FUNCTION IS_CTRL : BOOL
VAR_INPUT
	STR : STRING(STRING_LENGTH);
END_VAR
VAR
	L: INT;
	pt : POINTER TO BYTE;
	pos: INT;
END_VAR

(*
version 1.1	29. mar 2008
programmer 		kurt
tested by		hugo

IS_CTRL testet ob in einem string nur Steuerzeichen (Char < 32) vorkommen.

*)

PT := ADR(str);
L := LEN(str);
FOR pos := 1 TO L DO
	IF NOT (ISC_CTRL(pt^)) THEN
		IS_CTRL := FALSE;
		RETURN;
	END_IF;
    	PT := PT + 1;
END_FOR;
IS_CTRL := L > 0;


(* revision history
hm	29. feb. 2008	rev 1.0
	original version

hm	29. mar. 2008	rev 1.1
	changed STRING to STRING(STRING_LENGTH)
*)

END_FUNCTION

(* stored: Version 1.1.0.1, ProductVersion 3.1.4022.7
   POU IS_CTRL: Id {32bcadb6-541e-4a60-a3c1-23c6307ae02c}, SpecialFunc None *)
